PROGRAM SlaveArmControl
VAR
	// master robot data, input from master controller box
	m_masterRobotData AT %I* : MSCommu_MasterStatus;
	
	// all data from other tasks and controller 
	m_slaveInputDataPool : ST_SlaveInputDataPool;
		
	// slave robot data, ouput to master controller box
	m_slaveRobotData AT %Q* :MSCommu_slaveStatus;
	
	// slave robot status, including arm status and cartesian data, output to other tasks
	m_slaveStatus AT%Q* :ST_slaveStatus;
	
	// slave robot joint data, output to other tasks
	m_slaveJointsData AT %Q* :ST_slaveJointData;
	
	// flag to init robot
	m_robotInit :BOOL :=FALSE;
	
	// wait time before robot init  for ethercat to be statble 
	m_robotInitWaitTime : LREAL:=0;
	
	// slave robot
	m_slaveRobot:FB_SlaveRobot;

	// code execute time measure
	m_codeTime : Profiler;
	

END_VAR

m_codeTime(START:=TRUE, RESET:=TRUE);

// wait communication to be stable
IF(m_robotInitWaitTime<g_robotInitWaitTime) THEN
	m_robotInitWaitTime := m_robotInitWaitTime+g_slaveArmCtrlCycleTime;
	RETURN;
END_IF

// robot init
IF m_robotInit =FALSE THEN
	m_slaveRobot.Init();
	m_robotInit:=TRUE;
END_IF

// input from UI
UIInputProcess();

// master input data cast
masterInputDataCast(m_masterRobotData, m_slaveInputDataPool.m_masterStatus);

// robot run
m_slaveRobot.run(m_slaveInputDataPool);

// update data pool
m_slaveRobot.getStatus(m_slaveStatus,m_slaveJointsData);

// slave output data cast
slaveOutputDataCast(m_slaveInputDataPool.m_setupStatus, m_slaveStatus, m_slaveRobotData);

// output to UI
UIOutputProcess();

m_codeTime(START:=FALSE);

// convert from MSCommu_Mastertatus for master-slave communication to local ST_MasterStatus for control
METHOD masterInputDataCast : BOOL
VAR_IN_OUT CONSTANT
	masterInputData:MSCommu_MasterStatus;
END_VAR
VAR_IN_OUT
	masterStatus :ST_MasterStatus;
END_VAR

VAR
	i : INT;
END_VAR
masterStatus.m_masterHeartBeat := masterInputData.m_heartBeat;
masterStatus.m_motionScale := masterInputData.m_motionScale;
masterStatus.m_slaveSelfCheckFlag := masterInputData.m_slaveSelfCheckFlag;

FOR i:=1 TO g_mArmNum DO
	masterStatus.m_armState[i] := masterInputData.m_armState[i];
	masterStatus.m_teleSlaveArmIdx[i] :=masterInputData.m_teleSlaveArmIdx[i];
	masterStatus.m_gripAngle[i] := masterInputData.m_gripAngle[i];
	masterStatus.m_curArmPose[i].m_pos := masterInputData.m_curArmPose[i].m_pos;
	masterStatus.m_curArmPose[i].m_rot := masterInputData.m_curArmPose[i].m_rot;
	masterStatus.m_curArmTwist[i] :=masterInputData.m_curArmTwist[i];
END_FOR
END_METHOD

// convert from local ST_SlaveStatus for control to MSCommu_SlaveStatus for master-slave communication
METHOD slaveOutputDataCast : BOOL
VAR_IN_OUT CONSTANT
	setupStatus :ST_SetupStatus;
	slaveStatus :ST_SlaveStatus;
END_VAR
VAR_IN_OUT 
	slaveOutputData : MSCommu_SlaveStatus;
END_VAR

VAR
	slavePoseInCart, slavePoseInScope:ST_Frame;
	tmpFrame :ST_Frame;
	i :INT;
END_VAR
// Slave heart beat
IF slaveOutputData.m_heartBeat > 10 THEN
	slaveOutputData.m_heartBeat :=0;
ELSE
	slaveOutputData.m_heartBeat :=slaveOutputData.m_heartBeat+1;
END_IF

slaveOutputData.m_seflCheckPass:= slaveStatus.m_selfCheckPass[1] AND slaveStatus.m_selfCheckPass[2] AND slaveStatus.m_selfCheckPass[3] AND slaveStatus.m_selfCheckPass[4];

slaveOutputData.m_endoscopeMounted :=slaveStatus.m_endoscopeMounted;
slaveOutputData.m_endoscopePose.m_pos :=slaveStatus.m_endoscopePose.m_pos;
slaveOutputData.m_endoscopePose.m_rot :=slaveStatus.m_endoscopePose.m_rot;
FOR i:= 1 TO g_sArmNum DO
	slaveOutputData.m_armState[i] := slaveStatus.m_armState[i];
	slaveOutputData.m_instruStauts[i].m_fingerAngle := slaveStatus.m_instruStauts[i].m_fingerAngle;
	slaveOutputData.m_instruStauts[i].m_ready := slaveStatus.m_instruStauts[i].m_ready;
	slaveOutputData.m_instruStauts[i].m_type := slaveStatus.m_instruStauts[i].m_type;

	slavePoseInCart := transform(setupStatus.m_curEndPose[i], slaveStatus.m_curArmPose[i]);
	tmpFrame :=invFrame(slaveStatus.m_endoscopePose);
	slavePoseInScope := transform(tmpFrame, slavePoseInCart);
	slaveOutputData.m_curArmPose[i].m_pos :=slavePoseInScope.m_pos;
	slaveOutputData.m_curArmPose[i].m_rot :=slavePoseInScope.m_rot;
	slaveOutputData.m_masterSlavePoseError[i] :=slaveStatus.m_masterSlavePoseError[i];
END_FOR
END_METHOD

// tranform data from UI(global variable write by ADS) to ST_UIData
METHOD UIInputProcess : BOOL
VAR_INPUT
END_VAR
VAR
	i:int;
END_VAR
// arm disable
FOR i:=1 TO g_sArmNum DO 
	m_slaveInputDataPool.m_UIData.m_slaveArmDisableFlag[i]:= FALSE;
END_FOR
IF GVL_com_upper_PC.slaver_arm_disable >0 AND GVL_com_upper_PC.slaver_arm_disable<= g_sArmNum THEN
	m_slaveInputDataPool.m_UIData.m_slaveArmDisableFlag[GVL_com_upper_PC.slaver_arm_disable]:= TRUE;
END_IF
END_METHOD

METHOD UIOutputProcess : BOOL
VAR_INPUT
END_VAR
VAR
	i : INT;
END_VAR
//TODO
//control software version
GVL_com_upper_PC.version:='1(1.0.0.1)';

GVL_com_upper_PC.state_machine.Arm1_state_machine := m_slaveRobot.m_slaveArmState[1];
GVL_com_upper_PC.state_machine.Arm2_state_machine := m_slaveRobot.m_slaveArmState[2];
GVL_com_upper_PC.state_machine.Arm3_state_machine := m_slaveRobot.m_slaveArmState[3];
GVL_com_upper_PC.state_machine.Arm4_state_machine := m_slaveRobot.m_slaveArmState[4];
END_METHOD

END_PROGRAM

(* stored: Version 1.1.0.1, ProductVersion 3.1.4024.11
   POU SlaveArmControl: Id {6192c11b-cd6e-4883-b627-958acfb9caf3}, SpecialFunc None
   Method masterInputDataCast: Id {688f8323-8b5a-4cc7-b4b2-cb5f74424c3f}
   Method slaveOutputDataCast: Id {110717ec-abfc-4dc8-a3ed-d3c3fbcf321b}
   Method UIInputProcess: Id {9dd02246-5151-482e-a090-b6247e0a96d4}
   Method UIOutputProcess: Id {d0fa8c54-c1d5-4f7b-80a8-06c5ca1c6dd6} *)
